(* PLC project pulse_generator, Dassault Systèmes ControlBuild 2024x *)
(* stored: creationDateTime 2023-10-03T11:13:40-01:00 *)

FUNCTION_BLOCK bottling_line.pulse_generator
  VAR_INPUT
    speed : REAL := 0.0;
    sensorSupply : BOOL := true;
  END_VAR
  VAR_OUTPUT
    pulseSensor : BOOL := false;
  END_VAR
  VAR
    counter : REAL := 0.0;
  END_VAR
  VAR CONSTANT
    pulseDuration : REAL := 0.5;
  END_VAR
  VAR
    d_sensor : BOOL := false;
    v_d_sensor : BOOL := false;
  END_VAR


ACTION C_source_code:
/* -----------------------------------------------------------------------------------------------------------	*/
/* This module simulates the behaviour of a pulse generator		*/
/*	at the end of the conveyor belt.				*/
/* ----------------------------------------------------------------------------------------------------------	*/

if (d_sensor ) pulseSensor=v_d_sensor;
else
	if (( sensorSupply ) && (speed != 0.0)) {	
		counter += CLOCK_PERIOD/1000000.0;
		if (counter >= pulseDuration) {
			pulseSensor = ! pulseSensor;
			counter = 0.0;
		}
	}
	else pulseSensor = 0;
END_ACTION
END_FUNCTION_BLOCK
